// Mitsubishi GX Works2 project: X29   PLC: FX3G

// task Task_01 (event TRUE, interval 0, priority 31): POU_01

PROGRAM POU_01
VAR
  wstep : INT;
  ton1 : TON;
END_VAR
M99 := FALSE AND
M1 AND M2 AND M3 AND
Y0 AND Y1 AND Y2;

IF M8002 THEN
    wstep := 0;
END_IF;

IF NOT M0 THEN
    wstep := 0;
END_IF;

CASE wstep OF
    0:
        zrst(TRUE, Y0, Y2);
        ton1(in := FALSE);

        IF M1 THEN
            wstep := 20;
        END_IF;
        IF M2 THEN
            wstep := 40;
        END_IF;

    20:
        Y0 := TRUE;
        Y1 := (NOT M3) AND M2;
        Y2 := FALSE;
        ton1(in := NOT ton1.q, pt := t#10s);

        IF ton1.q THEN
        	M2 := FALSE;
        	M3 := FALSE;
            wstep := 0;
        END_IF;
    
    40:
        Y2 := TRUE;

        IF M1 THEN
            wstep := 20;
        END_IF;
END_CASE;
END_PROGRAM
